FUNCTION_BLOCK PUBLIC FB_DUT_HMI
VAR_INPUT
END_VAR
VAR_INPUT
    hmiValue_in: DUT_HMI;
END_VAR
VAR_OUTPUT
    hmiValue_out: DUT_HMI;
END_VAR
VAR
    intToBool: FB_Integer_To_BooleanArray;
    rbModeValues : ARRAY[0..1] OF BOOL;
	i: INT;
	ArrayLength: INT;
	OutputValue: INT;
	IntegerValue: INT;
END_VAR


//Convert HMI radioButton to BOOL
intToBool(IntegerValue:= hmiValue_in.ModeValue, ArrayLength:= 2);
hmiValue_out := hmiValue_in;
// Use BOOL array to set DUT_HMI values
rbModeValues := intToBool.OutputValue;	 
hmiValue_out.ManualOn := rbModeValues[0];
hmiValue_out.ManualOff := NOT rbModeValues[0];
hmiValue_out.AutoOn := rbModeValues[1];
hmiValue_out.AutoOff := NOT rbModeValues[1];

END_FUNCTION_BLOCK

(* stored: Version 1.1.0.1, ProductVersion 3.1.4024.12
   POU FB_DUT_HMI: Id {87d783e6-29d2-456c-9ea2-387c9cd56c88}, SpecialFunc None *)
